PROGRAM Drad_Internal
VAR
    fEncoderPosition : LREAL;
    EncoderPosition AT %Q* : DINT; //Encoder value for NC
    fScaler : LREAL := 100000;
END_VAR

GVL.astAxes[AXIS_DRAD_INTERNAL].stInputs.bLimitBwd := TRUE;
GVL.astAxes[AXIS_DRAD_INTERNAL].stInputs.bLimitFwd := TRUE;
GVL.astAxes[AXIS_DRAD_INTERNAL].stControl.bEnable := TRUE;

//E = SQRT(C^2 + F^2)


//calculate setpoint generator inputs
fEncoderPosition := SQRT(EXPT(astAxes[AXIS_DTANK_LENGTH].stStatus.fActPosition,2) + EXPT(astAxes[AXIS_DOFF_ANGLED].stStatus.fActPosition,2));
   
EncoderPosition:= LREAL_TO_DINT(fEncoderPosition * fScaler);

astAxes[AXIS_DRAD_INTERNAL].stDescription.sAxisName := 'DRAD_INTERNAL';

END_PROGRAM

(* stored: Version 1.1.0.1, ProductVersion 3.1.4024.12
   POU Drad_Internal: Id {9290ef43-cd17-453e-a826-bd93eb9f5add}, SpecialFunc None *)
